// TIA Portal V17 export
// export: Created 2024-08-09T12:53:23.6371835Z, ExportSetting WithDefaults, DisplayName Totally Integrated Automation Portal, DisplayVersion V17 Update 7, DisplayName TIA Portal Openness, DisplayVersion V17 Update 7, DisplayName TIA Portal Version Control Interface, DisplayVersion V17, DisplayName STEP 7 Professional, DisplayVersion V17 Update 7, DisplayName STEP 7 Safety, DisplayVersion V17 Update 6, DisplayName WinCC Professional, DisplayVersion V17 Update 7
TYPE "S_MODULE_SUIVI_COMMUNCHARG"
// stored: IsFailsafeCompliant false
   STRUCT
      Tab_Lots { ExternalAccessible := 'False'; ExternalVisible := 'False'; ExternalWritable := 'False'} : Array[0.."MAX_LOTS"] of "S_SuiviCommande";   // Table des zones de suivi lot
      NumLot { ExternalAccessible := 'False'; ExternalVisible := 'False'; ExternalWritable := 'False'} : USInt;   // no de lot pour gestion couleurs
      ArrCirPlein { ExternalAccessible := 'False'; ExternalVisible := 'False'; ExternalWritable := 'False'} : Bool;
   END_STRUCT;
END_TYPE
